PROGRAM P_Demo_DEC_TO_BCD
VAR
    fbDEC_TO_BCD : DEC_TO_BCD; // DEC_TO_BCD 实例
    START        : BOOL := FALSE;
    DIN          : BYTE := 0;
    BUSY         : BOOL;
    ERR          : BOOL;
    ERRID        : UDINT;
    BOUT         : BYTE;
END_VAR

// =============================================================================
// 场景：DEC_TO_BCD 的最小可编译演示——所有 VAR_INPUT 均以 doc/PDF 中真实引脚名调用。
//       业务侧请在线 monitor / 在线写值触发对应输入，看输出端 monitor 结果。
//
// 价值：保证示例 ST 代码所有引脚名与 DEC_TO_BCD 的 VAR_INPUT/VAR_OUTPUT 一致，
//       Add Existing Item (.TcPOU) → 编译 → 登录 流程能跑通，作为 hand-curated 例程
//       的脚手架。
//
// 验证步骤：
//   1. 引用 Tc2_Utilities（及其依赖 Tc2_System）
//   2. 右键 PLC 项目下 POUs 文件夹 → Add → Existing Item → 选本 .TcPOU 文件 → OK → 编译、登录
//   3. 在线对 VAR_INPUT 写入合适触发值（典型 bExecute / RUN / START 上升沿）
//   4. 在线 monitor VAR_OUTPUT 观察 FB 反应
// =============================================================================

fbDEC_TO_BCD(
    START := START,
    DIN := DIN,
    BUSY => BUSY,
    ERR => ERR,
    ERRID => ERRID,
    BOUT => BOUT
);

END_PROGRAM

(* stored: Version 1.1.0.1, ProductVersion 3.1.4024.5
   POU P_Demo_DEC_TO_BCD: Id {a4a5d7ca-90ab-5dba-b28a-05d313741eb5}, SpecialFunc None *)
